(* IEC 61131-3 sources: Elmo_Master/Lasal_PRG/MotionTCPDemo/Class/MotionControlIF, 1 file *)

(* ---- MotionControlIF.st ---- *)
(*!
<Class
	Name               = "MotionControlIF"
	Revision           = "0.0"
	RealtimeTask       = "true"
	CyclicTask         = "false"
	BackgroundTask     = "false"
	Sigmatek           = "false"
	OSInterface        = "false"
	HighPriority       = "false"
	Automatic          = "false"
	UpdateMode         = "Prescan"
	SharedCommandTable = "true"
	Objectsize         = "(388,0)">
	<Channels>
		<Server Name="ClassSvr" Visualized="false" Initialize="false" WriteProtected="true" Retentive="false"/>
		<Client Name="Axis4" Required="true" Internal="false"/>
		<Client Name="Axis5" Required="true" Internal="false"/>
		<Client Name="Axis6" Required="true" Internal="false"/>
		<Client Name="Axis7" Required="true" Internal="false"/>
		<Client Name="Axis8" Required="true" Internal="false"/>
		<Client Name="LMCProfil" Required="true" Internal="false"/>
		<Client Name="MAxis6_7_8" Required="true" Internal="false"/>
	</Channels>
	<Separators>
		<Clients>
			<SepChn Position="4"/>
		</Clients>
	</Separators>
</Class>
*)
MotionControlIF : CLASS
  //Servers:
	ClassSvr 	: SvrChCmd_DINT;
  //Clients:
	LMCProfil 	: CltChCmd__LMCProfile;
	Axis4 	: CltChCmd__LMCAxis;
	Axis5 	: CltChCmd__LMCAxis;
	MAxis6_7_8 	: CltChCmd__LMCAxis;
	Axis6 	: CltChCmd__LMCAxis;
	Axis7 	: CltChCmd__LMCAxis;
	Axis8 	: CltChCmd__LMCAxis;
  //Variables:
  //Functions:

	FUNCTION VIRTUAL GLOBAL RtWork
		VAR_INPUT
			EAX 	: UDINT;
		END_VAR
		VAR_OUTPUT
			state (EAX) 	: UDINT;
		END_VAR;
  //Tables:
	FUNCTION @STD
		VAR_OUTPUT
			ret_code	: CONFSTATES;
		END_VAR;
	FUNCTION GLOBAL TAB @CT_;
END_CLASS;

#pragma usingLtd _LMCAxis
#pragma usingLtd _LMCProfile

FUNCTION VIRTUAL GLOBAL MotionControlIF::RtWork
	VAR_INPUT
		EAX 	: UDINT;
	END_VAR
	VAR_OUTPUT
		state (EAX) 	: UDINT;
	END_VAR

	state := READY;

END_FUNCTION
